TYPE ST_Values_LineChart :
STRUCT
	x:LREAL;
	y:LREAL;

END_STRUCT
END_TYPE

(* stored: Version 1.1.0.1, ProductVersion 3.1.4022.6
   DUT ST_Values_LineChart: Id {49e12c2a-e5e1-4f76-ba1b-adef120a2bc8} *)
